Staubli VAL3: Day14.pjx

--- Day14.pjx ---
Parameters version=s8.13.1Cs9_BS2800 stackSize=5000 millimeterUnit=true
Program file=checkCombo.pgx
Program file=start.pgx
Program file=stop.pgx
Program file=unique.pgx
Data file=Day14.dtx
Library alias=util path=Disk://helpers/helpers.pjx
Library alias=math path=Disk://math/math.pjx
Library alias=str path=Disk://string/string.pjx
Library alias=stat path=Disk://statistics/statistics.pjx
Type name=lists path=Disk://types/lists/lists.pjx
Type name=lists_string_num path=Disk://types/lists_string_num/lists_string_num.pjx

--- Day14.dtx ---
string sInput
lists lResult
  [0]
    string sString
num nResult
string sStart
string sCombo[2]
string sResult
string sUnique
lists lSplit
  [0]
    string sString
lists_string_num lStrNum
  [0]
    string sString
    num nNum
num nUnique

--- start.pgx ---
program start()
  local num l_nElement
  local num l_nSplit
  local num l_nStep
  local num l_nLetter
  local num l_nMax
  local num l_nMin
begin

  // read file
  call util:readFile("Disk://input_day14.txt", sInput)
  // sInput[0] = "NNCB"

  // get the starting string
  sStart = sInput[0]

  // remove starting string and empty line
  delete(sInput[1])
  delete(sInput[0])

  call str:splitString(sInput," -> ", lResult)
  // lResult.sString[0] = "CH"
  // lResult.sString[1] = "B"

  // PUZZLE 1
  call str:splitWord(sStart, lSplit)

  // loop over all steps
  for l_nStep = 1 to 10
    resize(lStrNum,1,1)
    lStrNum.sString = ""
    lStrNum.nNum = -99
    for l_nSplit = size(lSplit.sString)-2 to 0 step -1

      sCombo[0] = lSplit.sString[l_nSplit]
      sCombo[1] = lSplit.sString[l_nSplit+1]

      call checkCombo(sResult)

      if sResult != ""
        append(lStrNum)
        lStrNum[size(lStrNum)-1].sString = sResult
        lStrNum[size(lStrNum)-1].nNum = l_nSplit+1
      endIf
    endFor

    // glue results together
    delete(lStrNum[0])
    for l_nElement = 0 to size(lStrNum)-1
      insert(lSplit.sString[lStrNum[l_nElement].nNum])
      lSplit.sString[lStrNum[l_nElement].nNum] = lStrNum[l_nElement].sString
    endFor

  endFor

  // get unique elements in result
  call unique(sUnique)
  resize(nUnique,1,1)
  nUnique[0] = 0
  resize(nUnique,1,size(sUnique))

  // calculate appearance of each unique element
  for l_nElement = 0 to size(lSplit.sString)-1
    for l_nLetter = 0 to size(sUnique)-1
      if lSplit.sString[l_nElement] == sUnique[l_nLetter]
        nUnique[l_nLetter] = nUnique[l_nLetter] +1
      endIf
    endFor
  endFor

  call util:max_(nUnique,l_nMax)
  call util:min_(nUnique,l_nMin)

  nResult = l_nMax-l_nMin
  call util:printNum(nResult)
  // 2447

end

--- checkCombo.pgx ---
program checkCombo(string& x_sResult)
  local num l_nCombo
begin

  for l_nCombo = 0 to size(lResult)-1

    if lResult[l_nCombo].sString == sCombo[0]+sCombo[1]

      x_sResult = lResult[l_nCombo].sString[1]
      return
    endIf

  endFor

  x_sResult = ""

end

--- unique.pgx ---
program unique(string& x_sResult[])
  local num l_nElement
  local bool l_bFound
  local num l_nBuffer
begin

  for l_nElement = 0 to size(lSplit.sString)-1
    l_bFound = false
    if l_nElement == 0
      append(x_sResult)
      x_sResult[size(x_sResult)-1] = lSplit.sString[l_nElement]
    else

      for l_nBuffer = 0 to size(x_sResult)-1
        if lSplit.sString[l_nElement] != x_sResult[l_nBuffer]
          l_bFound = false
        else
          // break out of for-loop
          l_bFound = true
          l_nBuffer = size(x_sResult)+1
        endIf

      endFor

      if l_bFound == false
        append(x_sResult)
        x_sResult[size(x_sResult)-1] = lSplit.sString[l_nElement]
      endIf

   endIf

  endFor

  delete(x_sResult[0])

end
